VAR_GLOBAL
	instRFIDInfeed	:	FactoryIO.FB_RFID;	//Instance of the RFID-Sensor
	finishedMessageReadSerialNumber	:	BOOL;
	reReadSerialNumber	:	R_TRIG;
	reFinishedMessageReadSerialNumber	:	R_TRIG;
	readData	:	DataPositions;
END_VAR

(* stored: Version 1.1.0.1
   GVL RFID: Id {c44171e8-d4bd-45d7-b43c-8561eeeb76b4} *)
